(* Logix 5000 project; controller SolisPLC_Vlad_CGL1 vendor 1 type 14 code 226 rev 32.13; software revision 32.02 *)

TASK MainTask (continuous, watchdog 500 ms) : MainProgram, DataLink, Palletizer
TASK SafetyTask (periodic, rate 20 ms, priority 10, watchdog 20 ms, safety) : SafetyProgram

MODULES
   Local : vendor 1 type 14 code 226 (5069 0, rev 32.13)
END_MODULES

TYPE UDT_MQTT_DINT :
STRUCT
   Message : DINT;
   Delay : DINT;
   Timer : TIMER;
   RawData : DINT;
   Delta : DINT;
   OldRawData : DINT;
END_STRUCT
END_TYPE

VAR_GLOBAL   (* controller tags *)
   MQTT_OUT : UDT_MQTT_DINT[100] := ([0].Message := 264, [0].Delay := -10000, [0].Timer.PRE := -10000, [0].Timer.ACC := 3160, [0].Timer.EN := 1, [0].Timer.TT := 1, [0].RawData := 264, [0].OldRawData := 264, [1].Message := 10, [1].RawData := 10, [1].OldRawData := 10, [2].Message := 12, [2].Delay := 100, [2].RawData := 16, [2].Delta := 5, [2].OldRawData := 12, [19].Timer.EN := 1, [19].Timer.TT := 1, [20].Timer.EN := 1, [20].Timer.TT := 1, [21].Timer.EN := 1, [21].Timer.TT := 1, [22].Timer.EN := 1, [22].Timer.TT := 1, [23].Timer.EN := 1, [23].Timer.TT := 1, [24].Timer.EN := 1, [24].Timer.TT := 1, [25].Timer.EN := 1, [25].Timer.TT := 1, [26].Timer.EN := 1, [26].Timer.TT := 1, [27].Timer.EN := 1, [27].Timer.TT := 1, [28].Timer.EN := 1, [28].Timer.TT := 1, [29].Timer.EN := 1, [29].Timer.TT := 1, [30].Timer.EN := 1, [30].Timer.TT := 1, [31].Timer.EN := 1, [31].Timer.TT := 1, [32].Timer.EN := 1, [32].Timer.TT := 1, [33].Timer.EN := 1, [33].Timer.TT := 1, [34].Timer.EN := 1, [34].Timer.TT := 1, [35].Timer.EN := 1, [35].Timer.TT := 1, [36].Timer.EN := 1, [36].Timer.TT := 1, [37].Timer.EN := 1, [37].Timer.TT := 1, [38].Timer.EN := 1, [38].Timer.TT := 1, [39].Timer.EN := 1, [39].Timer.DN := 1, [40].Timer.EN := 1, [40].Timer.DN := 1,
        [41].Timer.EN := 1, [41].Timer.DN := 1, [42].Timer.EN := 1, [42].Timer.DN := 1, [43].Timer.EN := 1, [43].Timer.DN := 1, [44].Timer.EN := 1, [44].Timer.DN := 1, [45].Timer.EN := 1, [45].Timer.DN := 1, [46].Timer.EN := 1, [46].Timer.DN := 1, [47].Timer.EN := 1, [47].Timer.DN := 1, [48].Timer.EN := 1, [48].Timer.DN := 1, [49].Timer.EN := 1, [49].Timer.DN := 1, [50].Timer.EN := 1, [50].Timer.DN := 1, [51].Timer.EN := 1, [51].Timer.DN := 1, [52].Timer.EN := 1, [52].Timer.DN := 1, [53].Timer.EN := 1, [53].Timer.DN := 1, [54].Timer.EN := 1, [54].Timer.DN := 1, [55].Timer.EN := 1, [55].Timer.DN := 1, [56].Timer.EN := 1, [56].Timer.DN := 1, [57].Timer.EN := 1, [57].Timer.DN := 1, [58].Timer.EN := 1, [58].Timer.DN := 1, [59].Timer.EN := 1, [59].Timer.DN := 1, [60].Timer.EN := 1, [60].Timer.DN := 1, [61].Timer.EN := 1, [61].Timer.DN := 1, [62].Timer.EN := 1, [62].Timer.DN := 1, [63].Timer.EN := 1, [63].Timer.DN := 1, [64].Timer.EN := 1, [64].Timer.DN := 1, [65].Timer.EN := 1, [65].Timer.DN := 1, [66].Timer.EN := 1, [66].Timer.DN := 1, [67].Timer.EN := 1, [67].Timer.DN := 1, [68].Timer.EN := 1, [68].Timer.DN := 1, [69].Timer.EN := 1, [69].Timer.DN := 1, [70].Timer.EN := 1, [70].Timer.DN := 1,
        [71].Timer.EN := 1, [71].Timer.DN := 1, [72].Timer.EN := 1, [72].Timer.DN := 1, [73].Timer.EN := 1, [73].Timer.DN := 1, [74].Timer.EN := 1, [74].Timer.DN := 1, [75].Timer.EN := 1, [75].Timer.DN := 1, [76].Timer.EN := 1, [76].Timer.DN := 1, [77].Timer.EN := 1, [77].Timer.DN := 1, [78].Timer.EN := 1, [78].Timer.DN := 1, [79].Timer.EN := 1, [79].Timer.DN := 1, [80].Timer.EN := 1, [80].Timer.DN := 1, [81].Timer.EN := 1, [81].Timer.DN := 1, [82].Timer.EN := 1, [82].Timer.DN := 1, [83].Timer.EN := 1, [83].Timer.DN := 1, [84].Timer.EN := 1, [84].Timer.DN := 1, [85].Timer.EN := 1, [85].Timer.DN := 1, [86].Timer.EN := 1, [86].Timer.DN := 1, [87].Timer.EN := 1, [87].Timer.DN := 1, [88].Timer.EN := 1, [88].Timer.DN := 1, [89].Timer.EN := 1, [89].Timer.DN := 1, [90].Timer.EN := 1, [90].Timer.DN := 1, [91].Timer.EN := 1, [91].Timer.DN := 1, [92].Timer.EN := 1, [92].Timer.DN := 1, [93].Timer.EN := 1, [93].Timer.DN := 1, [94].Timer.EN := 1, [94].Timer.DN := 1, [95].Timer.EN := 1, [95].Timer.DN := 1, [96].Timer.EN := 1, [96].Timer.DN := 1, [97].Timer.EN := 1, [97].Timer.TT := 1, [98].Timer.EN := 1, [98].Timer.TT := 1, [99].Timer.EN := 1, [99].Timer.TT := 1);
   MQTT_OUT_DINT : DINT[100] := ([0] := 4961, [1] := 4961, [2] := 4961);
   Pal_D : DINT[100] := ([0] := 264, [1] := 10, [2] := 16);
        [0].0   // Palletizer Infeed - Start PB
        [0].1   // Palletizer Infeed - Stop PB
        [0].10   // Palletizer Discharge - Stop PB
        [0].11   // Palletizer Discharge - Running Status
        [0].12   // Palletizer Discharge - Full Pallet Ready
        [0].2   // Palletizer Infeed - Enabled Status
        [0].3   // Palletizer Infeed - Full Status
        [0].4   // Palletizer Robot - Start PB
        [0].5   // Palletizer Robot - Stop PB
        [0].6   // Palletizer Robot - Enabled Status
        [0].7   // Palletizer Robot - Pick Up Cases
        [0].8   // Palletizer Robot - Cases On Arm
        [0].9   // Palletizer Discharge - Start PB
   Pal_T : TIMER[100] := ([0].PRE := 1000, [1].PRE := 4268, [2].PRE := 6639, [3].PRE := 7587);
   Sys_Timer : TIMER[100] := ([0].PRE := 100000, [0].ACC := 4976, [0].EN := 1, [0].TT := 1, [1].PRE := 500000, [1].ACC := 4976, [1].EN := 1, [1].TT := 1, [2].PRE := 11000, [2].ACC := 4976, [2].EN := 1, [2].TT := 1);
END_VAR

PROGRAM DataLink   (* main routine _01_Main *)
VAR
   index : DINT := 98;
END_VAR

ROUTINE _01_Main   (* ladder *)
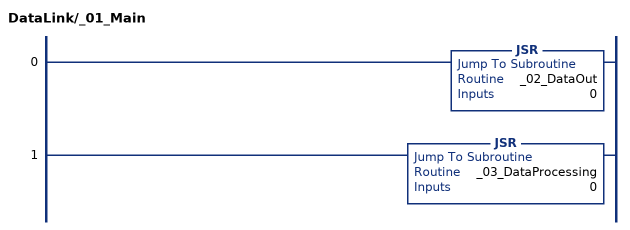
   0: JSR(_02_DataOut,0);
   1: JSR(_03_DataProcessing,0);
END_ROUTINE

ROUTINE _02_DataOut   (* ladder *)
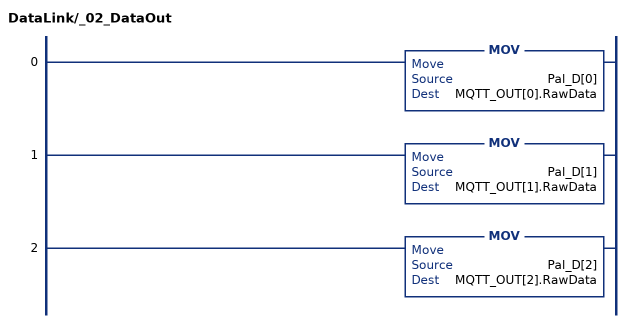
   0: MOV(Pal_D[0],MQTT_OUT[0].RawData);
   1: MOV(Pal_D[1],MQTT_OUT[1].RawData);
   2: MOV(Pal_D[2],MQTT_OUT[2].RawData);
END_ROUTINE

ROUTINE _03_DataProcessing   (* ladder *)
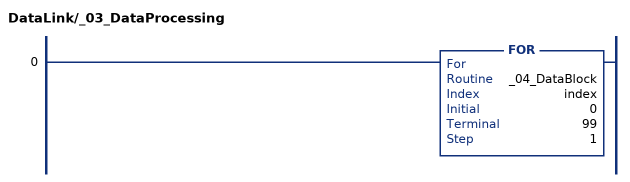
   0: FOR(_04_DataBlock,index,0,99,1);
END_ROUTINE

ROUTINE _04_DataBlock   (* ladder *)
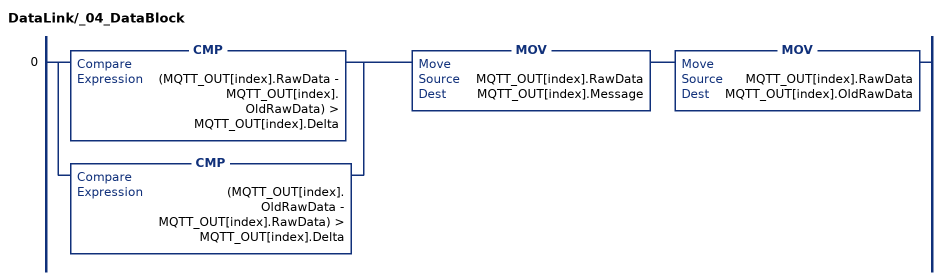
   0: [CMP((MQTT_OUT[index].RawData - MQTT_OUT[index].OldRawData) > MQTT_OUT[index].Delta) ,CMP((MQTT_OUT[index].OldRawData - MQTT_OUT[index].RawData) > MQTT_OUT[index].Delta) ]MOV(MQTT_OUT[index].RawData,MQTT_OUT[index].Message)MOV(MQTT_OUT[index].RawData,MQTT_OUT[index].OldRawData);
END_ROUTINE
END_PROGRAM

PROGRAM MainProgram   (* main routine MainRoutine *)

ROUTINE MainRoutine   (* ladder *)
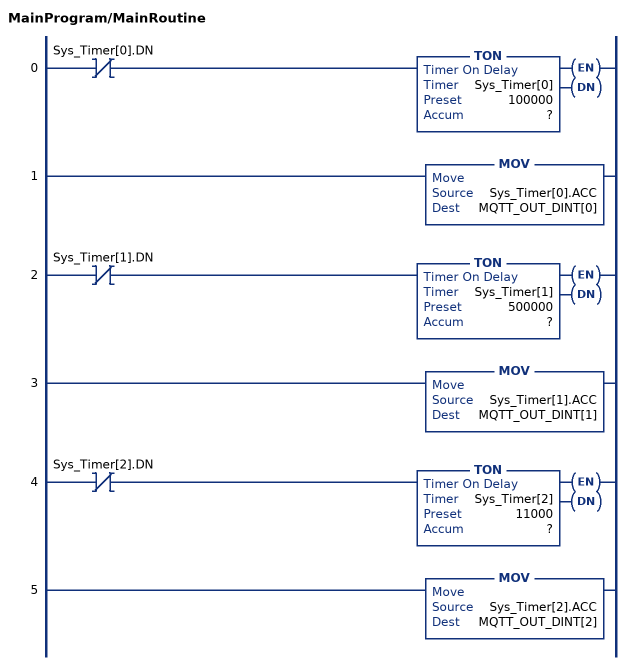
   0: XIO(Sys_Timer[0].DN)TON(Sys_Timer[0],?,?);
   1: MOV(Sys_Timer[0].ACC,MQTT_OUT_DINT[0]);
   2: XIO(Sys_Timer[1].DN)TON(Sys_Timer[1],?,?);
   3: MOV(Sys_Timer[1].ACC,MQTT_OUT_DINT[1]);
   4: XIO(Sys_Timer[2].DN)TON(Sys_Timer[2],?,?);
   5: MOV(Sys_Timer[2].ACC,MQTT_OUT_DINT[2]);
END_ROUTINE
END_PROGRAM

PROGRAM Palletizer   (* main routine _01_Main *)
VAR
   Mask : DINT[20];
   Mask1 : DINT;
   RandomNum : DINT := 14705320;
   ScanTime : DINT := 127;
   Time : DINT[7] := ([0] := 1998, [1] := 12, [2] := 28, [4] := 14, [5] := 41, [6] := 477906);
END_VAR

ROUTINE _01_Main   (* ladder *)
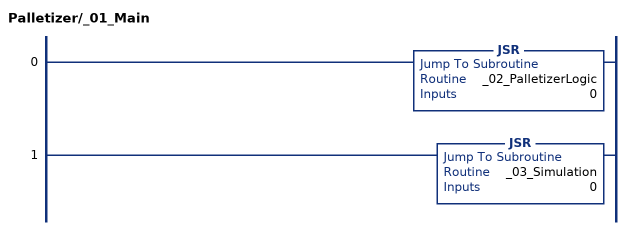
   0: JSR(_02_PalletizerLogic,0);
   1: JSR(_03_Simulation,0);
END_ROUTINE

ROUTINE _02_PalletizerLogic   (* ladder *)
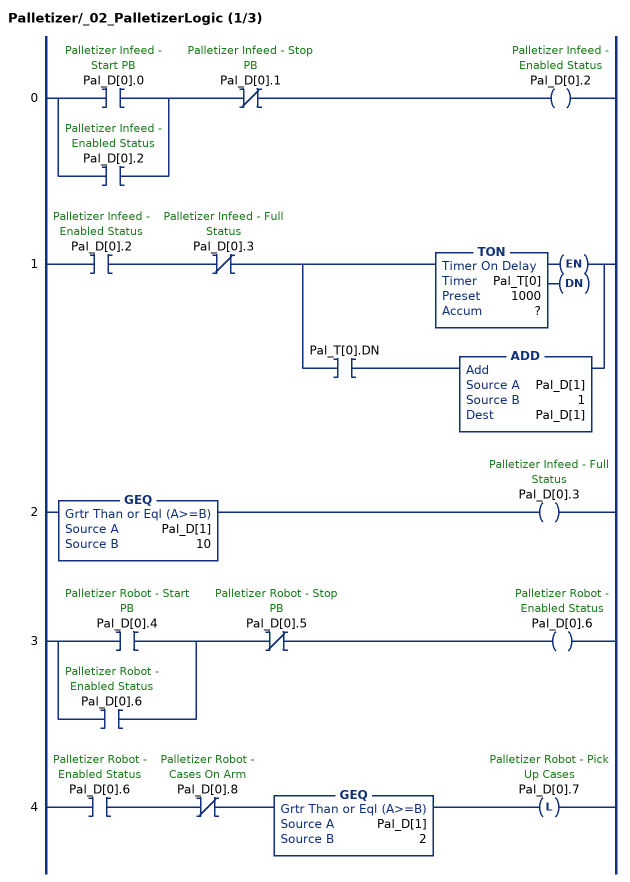
   0: [XIC(Pal_D[0].0) ,XIC(Pal_D[0].2) ]XIO(Pal_D[0].1)OTE(Pal_D[0].2);
   1: XIC(Pal_D[0].2)XIO(Pal_D[0].3)[TON(Pal_T[0],?,?) ,XIC(Pal_T[0].DN) ADD(Pal_D[1],1,Pal_D[1]) ];
   2: GEQ(Pal_D[1],10)OTE(Pal_D[0].3);
   3: [XIC(Pal_D[0].4) ,XIC(Pal_D[0].6) ]XIO(Pal_D[0].5)OTE(Pal_D[0].6);
   4: XIC(Pal_D[0].6)XIO(Pal_D[0].8)GEQ(Pal_D[1],2)OTL(Pal_D[0].7);
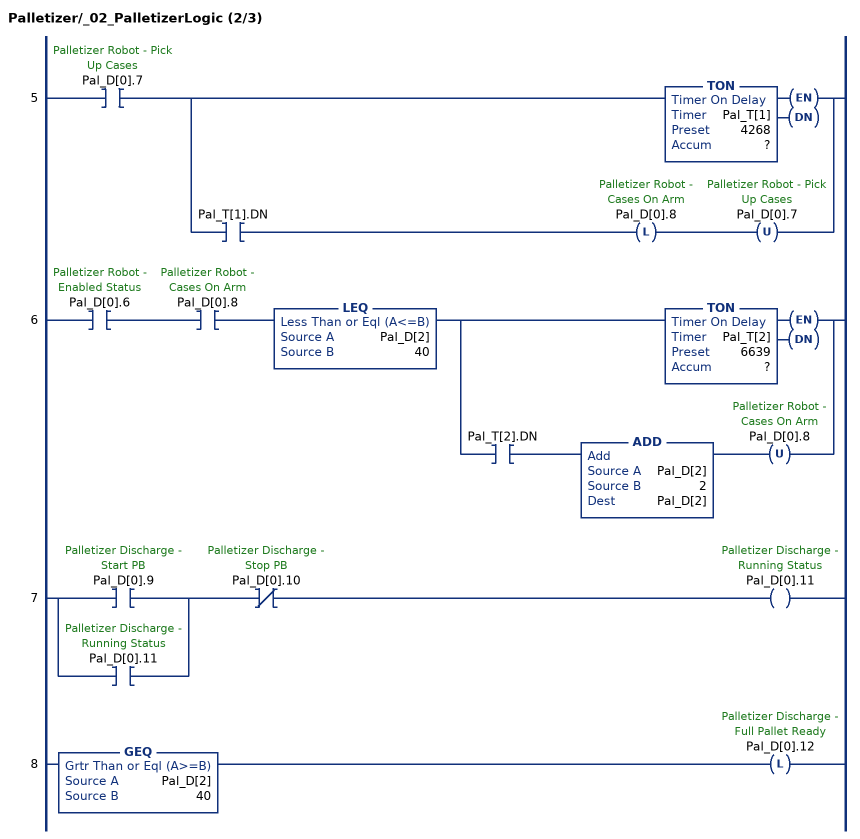
   5: XIC(Pal_D[0].7)[TON(Pal_T[1],?,?) ,XIC(Pal_T[1].DN) OTL(Pal_D[0].8) OTU(Pal_D[0].7) ];
   6: XIC(Pal_D[0].6)XIC(Pal_D[0].8)LEQ(Pal_D[2],40)[TON(Pal_T[2],?,?) ,XIC(Pal_T[2].DN) ADD(Pal_D[2],2,Pal_D[2]) OTU(Pal_D[0].8) ];
   7: [XIC(Pal_D[0].9) ,XIC(Pal_D[0].11) ]XIO(Pal_D[0].10)OTE(Pal_D[0].11);
   8: GEQ(Pal_D[2],40)OTL(Pal_D[0].12);
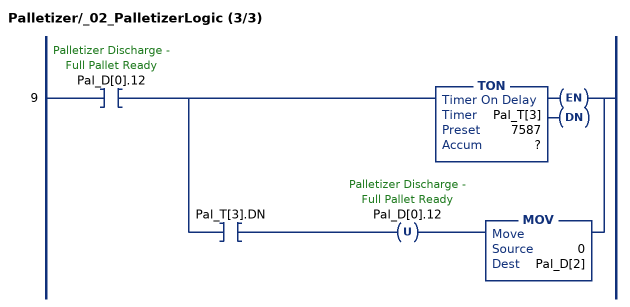
   9: XIC(Pal_D[0].12)[TON(Pal_T[3],?,?) ,XIC(Pal_T[3].DN) OTU(Pal_D[0].12) MOV(0,Pal_D[2]) ];
END_ROUTINE

ROUTINE _03_Simulation   (* ladder *)
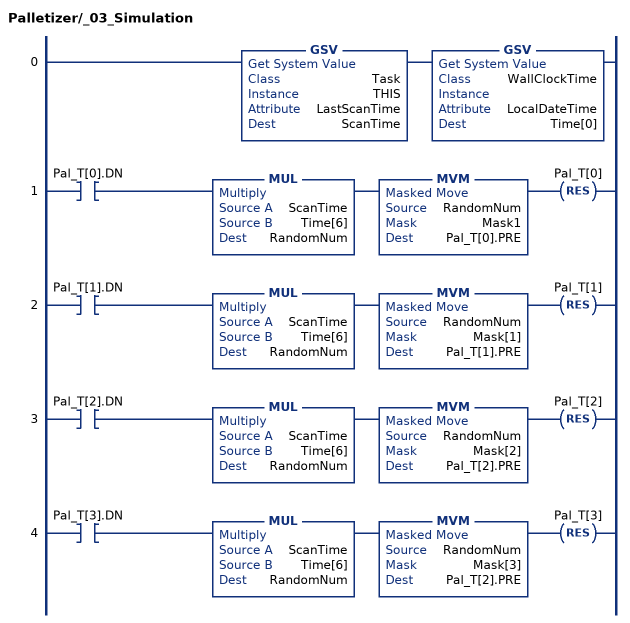
   0: GSV(Task,THIS,LastScanTime,ScanTime)GSV(WallClockTime,,LocalDateTime,Time[0]);
   1: XIC(Pal_T[0].DN)MUL(ScanTime,Time[6],RandomNum)MVM(RandomNum,Mask1,Pal_T[0].PRE)RES(Pal_T[0]);
   2: XIC(Pal_T[1].DN)MUL(ScanTime,Time[6],RandomNum)MVM(RandomNum,Mask[1],Pal_T[1].PRE)RES(Pal_T[1]);
   3: XIC(Pal_T[2].DN)MUL(ScanTime,Time[6],RandomNum)MVM(RandomNum,Mask[2],Pal_T[2].PRE)RES(Pal_T[2]);
   4: XIC(Pal_T[3].DN)MUL(ScanTime,Time[6],RandomNum)MVM(RandomNum,Mask[3],Pal_T[2].PRE)RES(Pal_T[3]);
END_ROUTINE
END_PROGRAM

PROGRAM SafetyProgram   (* main routine MainRoutine, safety *)

ROUTINE MainRoutine   (* ladder *)
END_ROUTINE
END_PROGRAM
